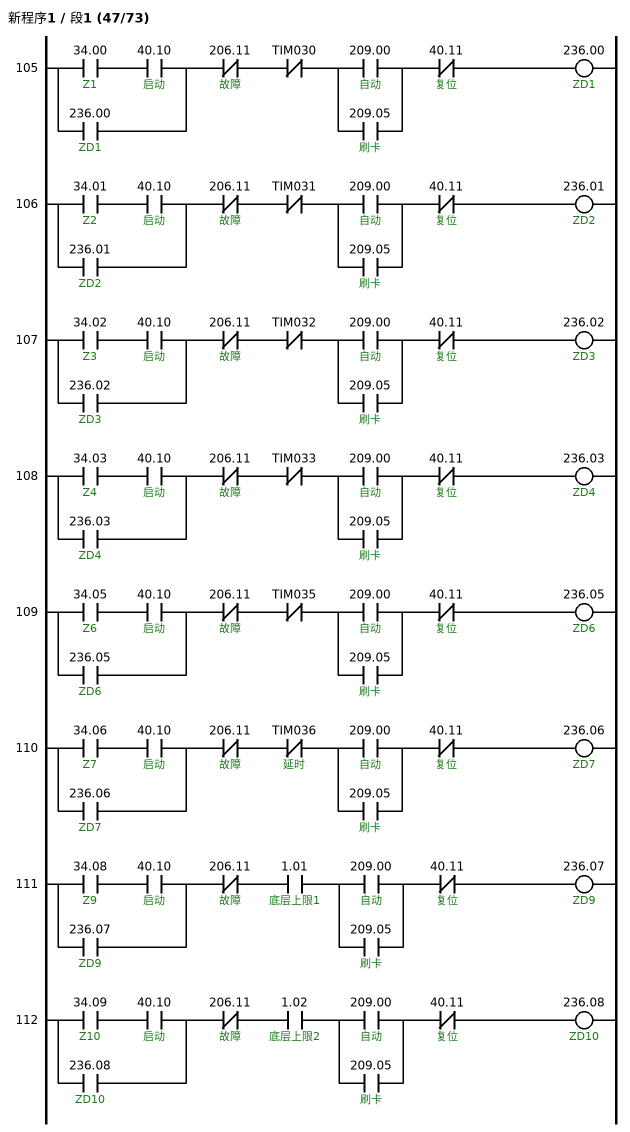
; [picture p48: 新程序1 / 段1, rungs 105-112]
; rung 105
LD 34.00  ; Z1
AND 40.10  ; 启动
OR 236.00  ; ZD1
ANDNOT 206.11  ; 故障
ANDNOT TIM030
LD 209.00  ; 自动
OR 209.05  ; 刷卡
ANDLD
ANDNOT 40.11  ; 复位
OUT 236.00  ; ZD1
; rung 106
LD 34.01  ; Z2
AND 40.10  ; 启动
OR 236.01  ; ZD2
ANDNOT 206.11  ; 故障
ANDNOT TIM031
LD 209.00  ; 自动
OR 209.05  ; 刷卡
ANDLD
ANDNOT 40.11  ; 复位
OUT 236.01  ; ZD2
; rung 107
LD 34.02  ; Z3
AND 40.10  ; 启动
OR 236.02  ; ZD3
ANDNOT 206.11  ; 故障
ANDNOT TIM032
LD 209.00  ; 自动
OR 209.05  ; 刷卡
ANDLD
ANDNOT 40.11  ; 复位
OUT 236.02  ; ZD3
; rung 108
LD 34.03  ; Z4
AND 40.10  ; 启动
OR 236.03  ; ZD4
ANDNOT 206.11  ; 故障
ANDNOT TIM033
LD 209.00  ; 自动
OR 209.05  ; 刷卡
ANDLD
ANDNOT 40.11  ; 复位
OUT 236.03  ; ZD4
; rung 109
LD 34.05  ; Z6
AND 40.10  ; 启动
OR 236.05  ; ZD6
ANDNOT 206.11  ; 故障
ANDNOT TIM035
LD 209.00  ; 自动
OR 209.05  ; 刷卡
ANDLD
ANDNOT 40.11  ; 复位
OUT 236.05  ; ZD6
; rung 110
LD 34.06  ; Z7
AND 40.10  ; 启动
OR 236.06  ; ZD7
ANDNOT 206.11  ; 故障
ANDNOT TIM036  ; 延时
LD 209.00  ; 自动
OR 209.05  ; 刷卡
ANDLD
ANDNOT 40.11  ; 复位
OUT 236.06  ; ZD7
; rung 111
LD 34.08  ; Z9
AND 40.10  ; 启动
OR 236.07  ; ZD9
ANDNOT 206.11  ; 故障
AND 1.01  ; 底层上限1
LD 209.00  ; 自动
OR 209.05  ; 刷卡
ANDLD
ANDNOT 40.11  ; 复位
OUT 236.07  ; ZD9
; rung 112
LD 34.09  ; Z10
AND 40.10  ; 启动
OR 236.08  ; ZD10
ANDNOT 206.11  ; 故障
AND 1.02  ; 底层上限2
LD 209.00  ; 自动
OR 209.05  ; 刷卡
ANDLD
ANDNOT 40.11  ; 复位
OUT 236.08  ; ZD10

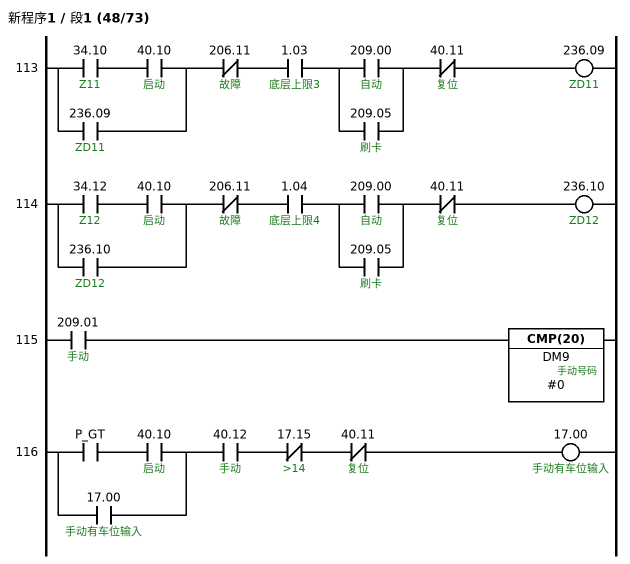
; rung 113
LD 34.10  ; Z11
AND 40.10  ; 启动
OR 236.09  ; ZD11
ANDNOT 206.11  ; 故障
AND 1.03  ; 底层上限3
LD 209.00  ; 自动
OR 209.05  ; 刷卡
ANDLD
ANDNOT 40.11  ; 复位
OUT 236.09  ; ZD11
; rung 114
LD 34.12  ; Z12
AND 40.10  ; 启动
OR 236.10  ; ZD12
ANDNOT 206.11  ; 故障
AND 1.04  ; 底层上限4
LD 209.00  ; 自动
OR 209.05  ; 刷卡
ANDLD
ANDNOT 40.11  ; 复位
OUT 236.10  ; ZD12
; rung 115
LD 209.01  ; 手动
CMP(20) DM9 #0  ; 手动号码
; rung 116
LD P_GT
AND 40.10  ; 启动
OR 17.00  ; 手动有车位输入
AND 40.12  ; 手动
ANDNOT 17.15  ; >14
ANDNOT 40.11  ; 复位
OUT 17.00  ; 手动有车位输入

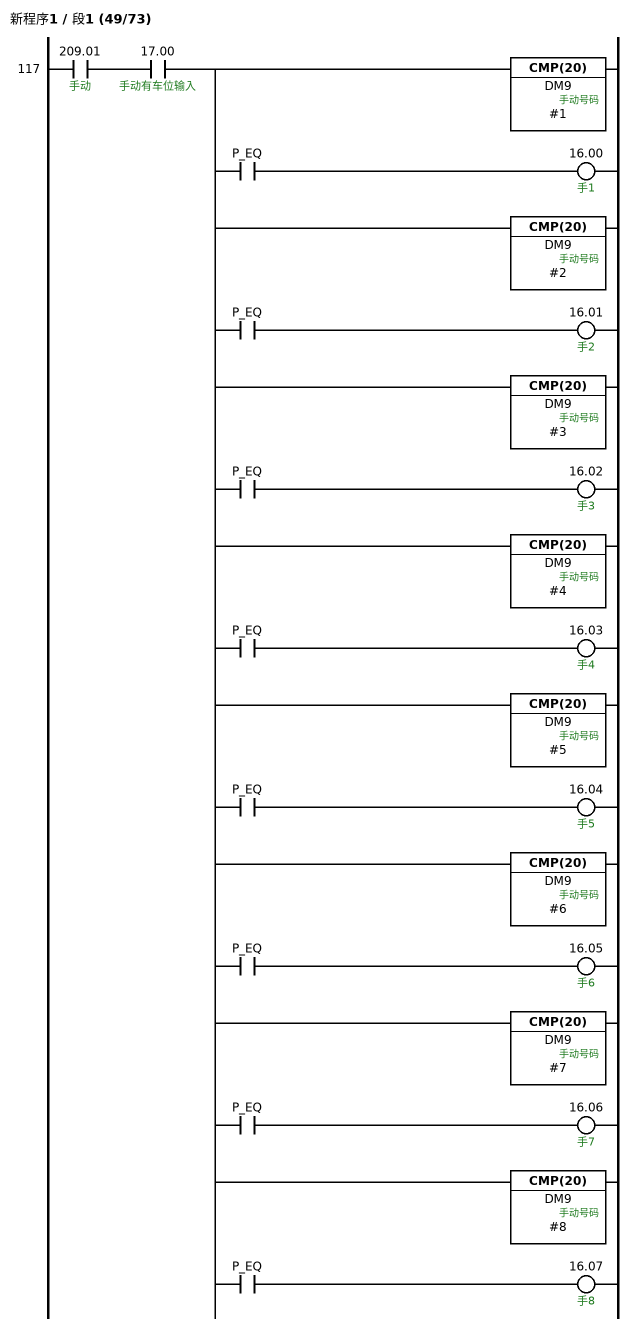

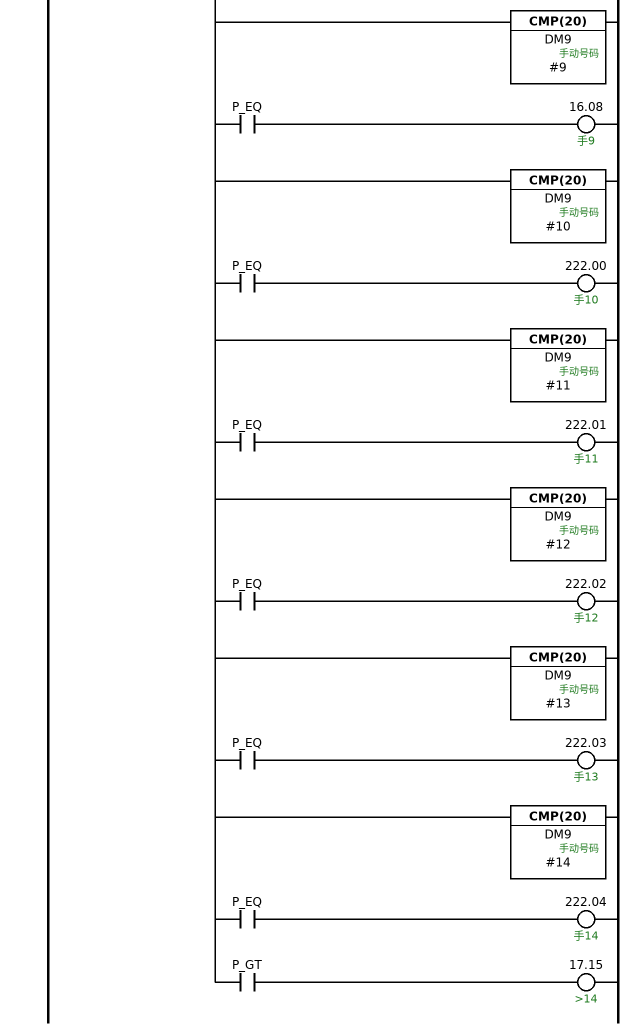
; rung 117
LD 209.01  ; 手动
AND 17.00  ; 手动有车位输入
OUT TR0
CMP(20) DM9 #1  ; 手动号码
AND P_EQ
OUT 16.00  ; 手1
LD TR0
CMP(20) DM9 #2  ; 手动号码
AND P_EQ
OUT 16.01  ; 手2
LD TR0
CMP(20) DM9 #3  ; 手动号码
AND P_EQ
OUT 16.02  ; 手3
LD TR0
CMP(20) DM9 #4  ; 手动号码
AND P_EQ
OUT 16.03  ; 手4
LD TR0
CMP(20) DM9 #5  ; 手动号码
AND P_EQ
OUT 16.04  ; 手5
LD TR0
CMP(20) DM9 #6  ; 手动号码
AND P_EQ
OUT 16.05  ; 手6
LD TR0
CMP(20) DM9 #7  ; 手动号码
AND P_EQ
OUT 16.06  ; 手7
LD TR0
CMP(20) DM9 #8  ; 手动号码
AND P_EQ
OUT 16.07  ; 手8
LD TR0
CMP(20) DM9 #9  ; 手动号码
AND P_EQ
OUT 16.08  ; 手9
LD TR0
CMP(20) DM9 #10  ; 手动号码
AND P_EQ
OUT 222.00  ; 手10
LD TR0
CMP(20) DM9 #11  ; 手动号码
AND P_EQ
OUT 222.01  ; 手11
LD TR0
CMP(20) DM9 #12  ; 手动号码
AND P_EQ
OUT 222.02  ; 手12
LD TR0
CMP(20) DM9 #13  ; 手动号码
AND P_EQ
OUT 222.03  ; 手13
LD TR0
CMP(20) DM9 #14  ; 手动号码
AND P_EQ
OUT 222.04  ; 手14
LD TR0
AND P_GT
OUT 17.15  ; >14

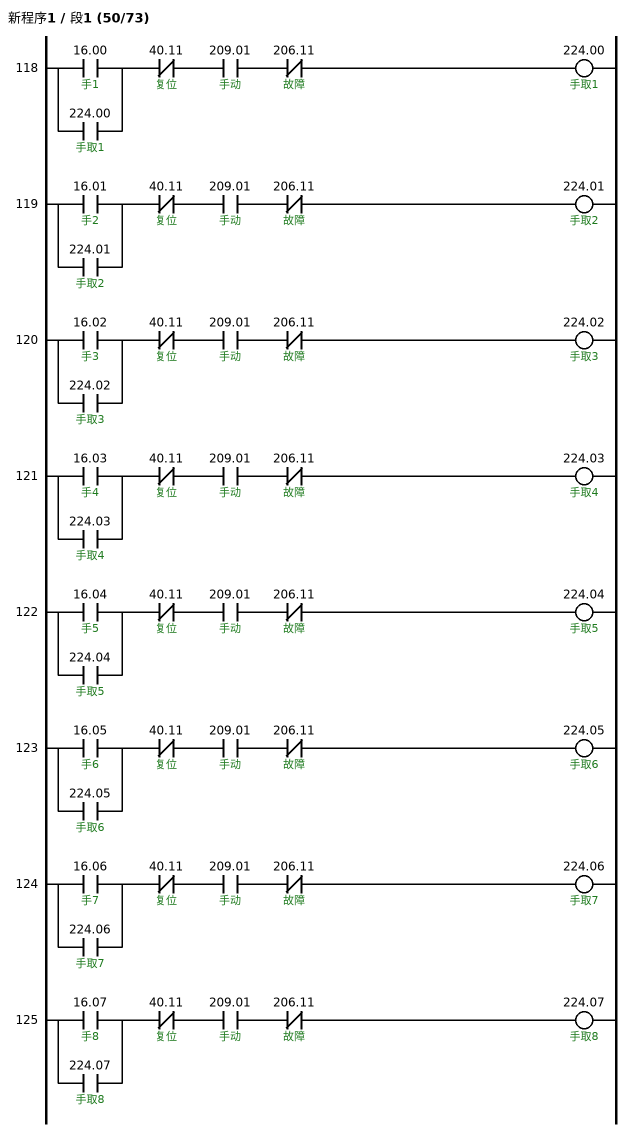
; rung 118
LD 16.00  ; 手1
OR 224.00  ; 手取1
ANDNOT 40.11  ; 复位
AND 209.01  ; 手动
ANDNOT 206.11  ; 故障
OUT 224.00  ; 手取1
; rung 119
LD 16.01  ; 手2
OR 224.01  ; 手取2
ANDNOT 40.11  ; 复位
AND 209.01  ; 手动
ANDNOT 206.11  ; 故障
OUT 224.01  ; 手取2
; rung 120
LD 16.02  ; 手3
OR 224.02  ; 手取3
ANDNOT 40.11  ; 复位
AND 209.01  ; 手动
ANDNOT 206.11  ; 故障
OUT 224.02  ; 手取3
; rung 121
LD 16.03  ; 手4
OR 224.03  ; 手取4
ANDNOT 40.11  ; 复位
AND 209.01  ; 手动
ANDNOT 206.11  ; 故障
OUT 224.03  ; 手取4
; rung 122
LD 16.04  ; 手5
OR 224.04  ; 手取5
ANDNOT 40.11  ; 复位
AND 209.01  ; 手动
ANDNOT 206.11  ; 故障
OUT 224.04  ; 手取5
; rung 123
LD 16.05  ; 手6
OR 224.05  ; 手取6
ANDNOT 40.11  ; 复位
AND 209.01  ; 手动
ANDNOT 206.11  ; 故障
OUT 224.05  ; 手取6
; rung 124
LD 16.06  ; 手7
OR 224.06  ; 手取7
ANDNOT 40.11  ; 复位
AND 209.01  ; 手动
ANDNOT 206.11  ; 故障
OUT 224.06  ; 手取7
; rung 125
LD 16.07  ; 手8
OR 224.07  ; 手取8
ANDNOT 40.11  ; 复位
AND 209.01  ; 手动
ANDNOT 206.11  ; 故障
OUT 224.07  ; 手取8

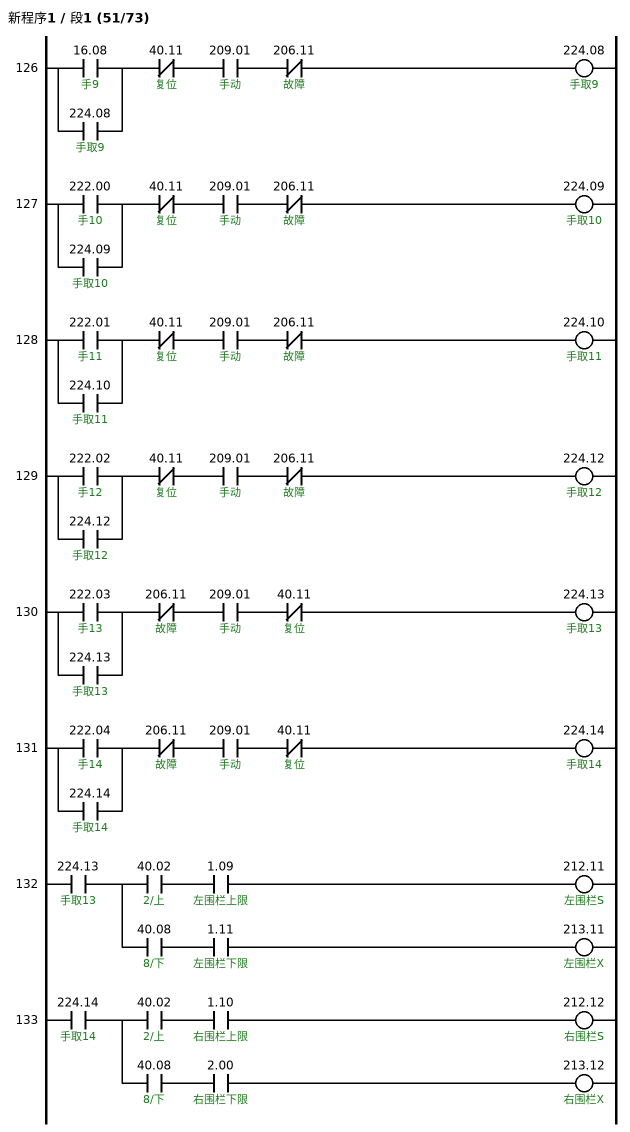
; rung 126
LD 16.08  ; 手9
OR 224.08  ; 手取9
ANDNOT 40.11  ; 复位
AND 209.01  ; 手动
ANDNOT 206.11  ; 故障
OUT 224.08  ; 手取9
; rung 127
LD 222.00  ; 手10
OR 224.09  ; 手取10
ANDNOT 40.11  ; 复位
AND 209.01  ; 手动
ANDNOT 206.11  ; 故障
OUT 224.09  ; 手取10
; rung 128
LD 222.01  ; 手11
OR 224.10  ; 手取11
ANDNOT 40.11  ; 复位
AND 209.01  ; 手动
ANDNOT 206.11  ; 故障
OUT 224.10  ; 手取11
; rung 129
LD 222.02  ; 手12
OR 224.12  ; 手取12
ANDNOT 40.11  ; 复位
AND 209.01  ; 手动
ANDNOT 206.11  ; 故障
OUT 224.12  ; 手取12
; rung 130
LD 222.03  ; 手13
OR 224.13  ; 手取13
ANDNOT 206.11  ; 故障
AND 209.01  ; 手动
ANDNOT 40.11  ; 复位
OUT 224.13  ; 手取13
; rung 131
LD 222.04  ; 手14
OR 224.14  ; 手取14
ANDNOT 206.11  ; 故障
AND 209.01  ; 手动
ANDNOT 40.11  ; 复位
OUT 224.14  ; 手取14
; rung 132
LD 224.13  ; 手取13
OUT TR0
AND 40.02  ; 2/上
AND 1.09  ; 左围栏上限
OUT 212.11  ; 左围栏S
LD TR0
AND 40.08  ; 8/下
AND 1.11  ; 左围栏下限
OUT 213.11  ; 左围栏X
; rung 133
LD 224.14  ; 手取14
OUT TR0
AND 40.02  ; 2/上
AND 1.10  ; 右围栏上限
OUT 212.12  ; 右围栏S
LD TR0
AND 40.08  ; 8/下
AND 2.00  ; 右围栏下限
OUT 213.12  ; 右围栏X

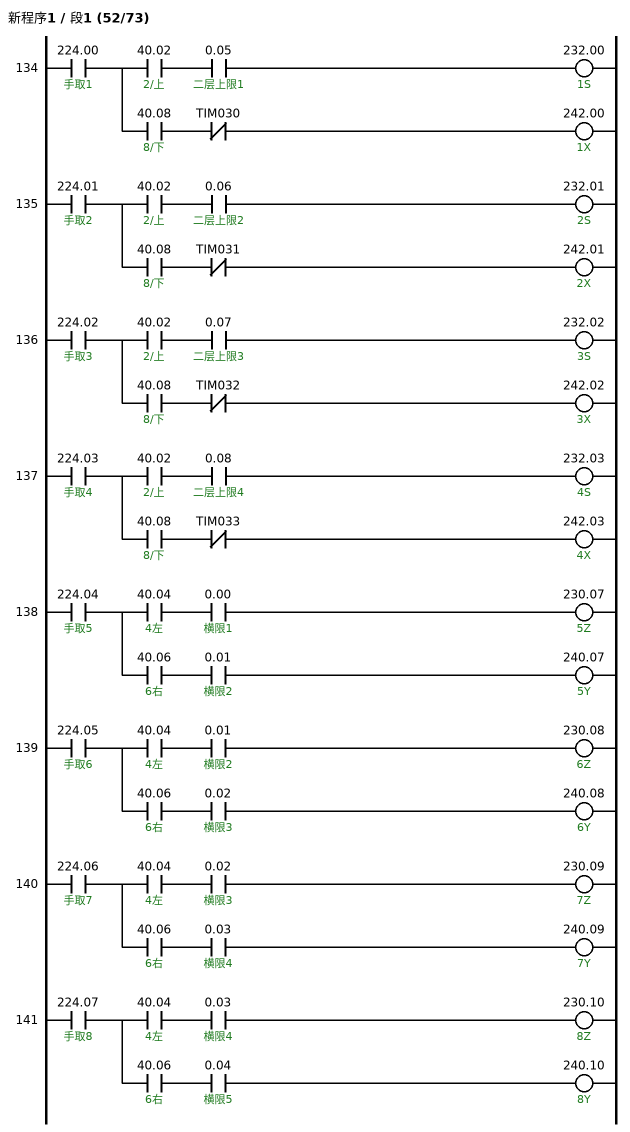
; rung 134
LD 224.00  ; 手取1
OUT TR0
AND 40.02  ; 2/上
AND 0.05  ; 二层上限1
OUT 232.00  ; 1S
LD TR0
AND 40.08  ; 8/下
ANDNOT TIM030
OUT 242.00  ; 1X
; rung 135
LD 224.01  ; 手取2
OUT TR0
AND 40.02  ; 2/上
AND 0.06  ; 二层上限2
OUT 232.01  ; 2S
LD TR0
AND 40.08  ; 8/下
ANDNOT TIM031
OUT 242.01  ; 2X
; rung 136
LD 224.02  ; 手取3
OUT TR0
AND 40.02  ; 2/上
AND 0.07  ; 二层上限3
OUT 232.02  ; 3S
LD TR0
AND 40.08  ; 8/下
ANDNOT TIM032
OUT 242.02  ; 3X
; rung 137
LD 224.03  ; 手取4
OUT TR0
AND 40.02  ; 2/上
AND 0.08  ; 二层上限4
OUT 232.03  ; 4S
LD TR0
AND 40.08  ; 8/下
ANDNOT TIM033
OUT 242.03  ; 4X
; rung 138
LD 224.04  ; 手取5
OUT TR0
AND 40.04  ; 4左
AND 0.00  ; 横限1
OUT 230.07  ; 5Z
LD TR0
AND 40.06  ; 6右
AND 0.01  ; 横限2
OUT 240.07  ; 5Y
; rung 139
LD 224.05  ; 手取6
OUT TR0
AND 40.04  ; 4左
AND 0.01  ; 横限2
OUT 230.08  ; 6Z
LD TR0
AND 40.06  ; 6右
AND 0.02  ; 横限3
OUT 240.08  ; 6Y
; rung 140
LD 224.06  ; 手取7
OUT TR0
AND 40.04  ; 4左
AND 0.02  ; 横限3
OUT 230.09  ; 7Z
LD TR0
AND 40.06  ; 6右
AND 0.03  ; 横限4
OUT 240.09  ; 7Y
; rung 141
LD 224.07  ; 手取8
OUT TR0
AND 40.04  ; 4左
AND 0.03  ; 横限4
OUT 230.10  ; 8Z
LD TR0
AND 40.06  ; 6右
AND 0.04  ; 横限5
OUT 240.10  ; 8Y

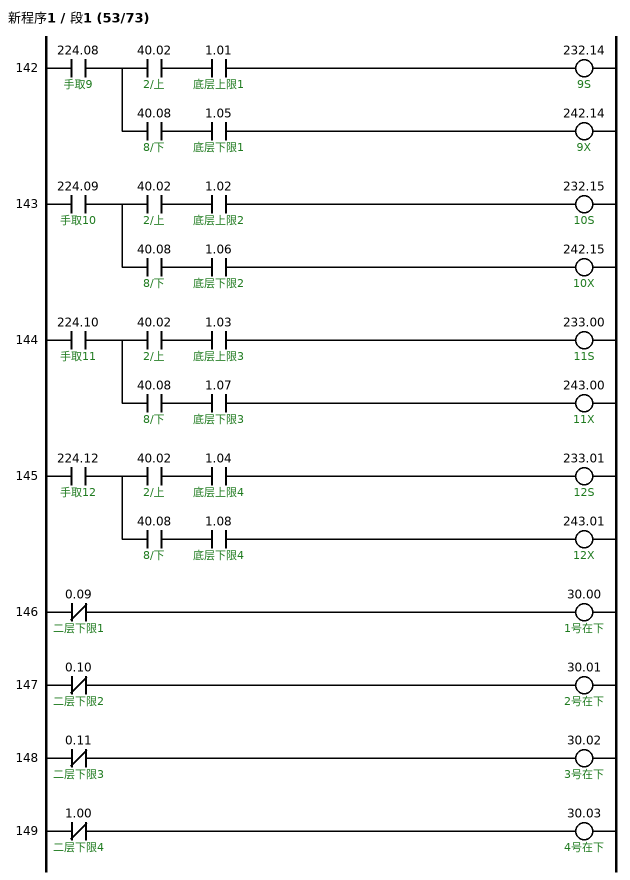
; rung 142
LD 224.08  ; 手取9
OUT TR0
AND 40.02  ; 2/上
AND 1.01  ; 底层上限1
OUT 232.14  ; 9S
LD TR0
AND 40.08  ; 8/下
AND 1.05  ; 底层下限1
OUT 242.14  ; 9X
; rung 143
LD 224.09  ; 手取10
OUT TR0
AND 40.02  ; 2/上
AND 1.02  ; 底层上限2
OUT 232.15  ; 10S
LD TR0
AND 40.08  ; 8/下
AND 1.06  ; 底层下限2
OUT 242.15  ; 10X
; rung 144
LD 224.10  ; 手取11
OUT TR0
AND 40.02  ; 2/上
AND 1.03  ; 底层上限3
OUT 233.00  ; 11S
LD TR0
AND 40.08  ; 8/下
AND 1.07  ; 底层下限3
OUT 243.00  ; 11X
; rung 145
LD 224.12  ; 手取12
OUT TR0
AND 40.02  ; 2/上
AND 1.04  ; 底层上限4
OUT 233.01  ; 12S
LD TR0
AND 40.08  ; 8/下
AND 1.08  ; 底层下限4
OUT 243.01  ; 12X
; rung 146
LDNOT 0.09  ; 二层下限1
OUT 30.00  ; 1号在下
; rung 147
LDNOT 0.10  ; 二层下限2
OUT 30.01  ; 2号在下
; rung 148
LDNOT 0.11  ; 二层下限3
OUT 30.02  ; 3号在下
; rung 149
LDNOT 1.00  ; 二层下限4
OUT 30.03  ; 4号在下

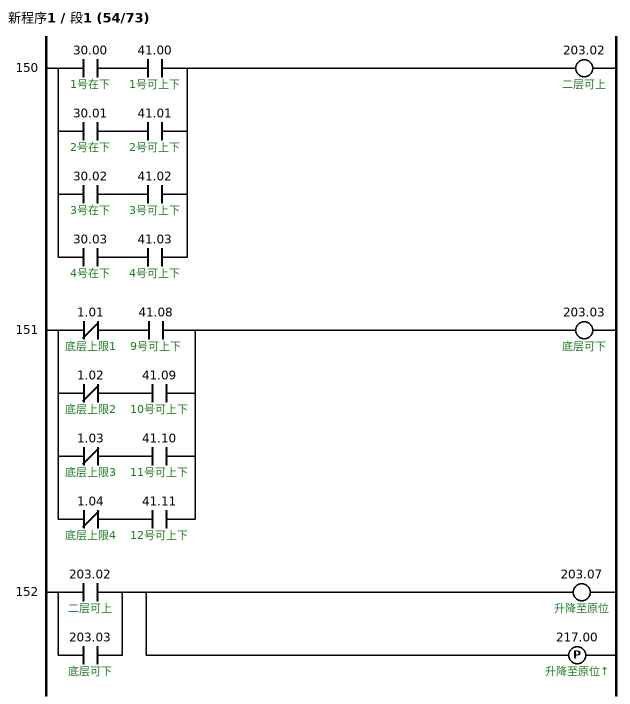
; rung 150
LD 30.00  ; 1号在下
AND 41.00  ; 1号可上下
LD 30.01  ; 2号在下
AND 41.01  ; 2号可上下
ORLD
LD 30.02  ; 3号在下
AND 41.02  ; 3号可上下
ORLD
LD 30.03  ; 4号在下
AND 41.03  ; 4号可上下
ORLD
OUT 203.02  ; 二层可上
; rung 151
LDNOT 1.01  ; 底层上限1
AND 41.08  ; 9号可上下
LDNOT 1.02  ; 底层上限2
AND 41.09  ; 10号可上下
ORLD
LDNOT 1.03  ; 底层上限3
AND 41.10  ; 11号可上下
ORLD
LDNOT 1.04  ; 底层上限4
AND 41.11  ; 12号可上下
ORLD
OUT 203.03  ; 底层可下
; rung 152
LD 203.02  ; 二层可上
OR 203.03  ; 底层可下
OUT 203.07  ; 升降至原位
DIFU(13) 217.00  ; 升降至原位↑

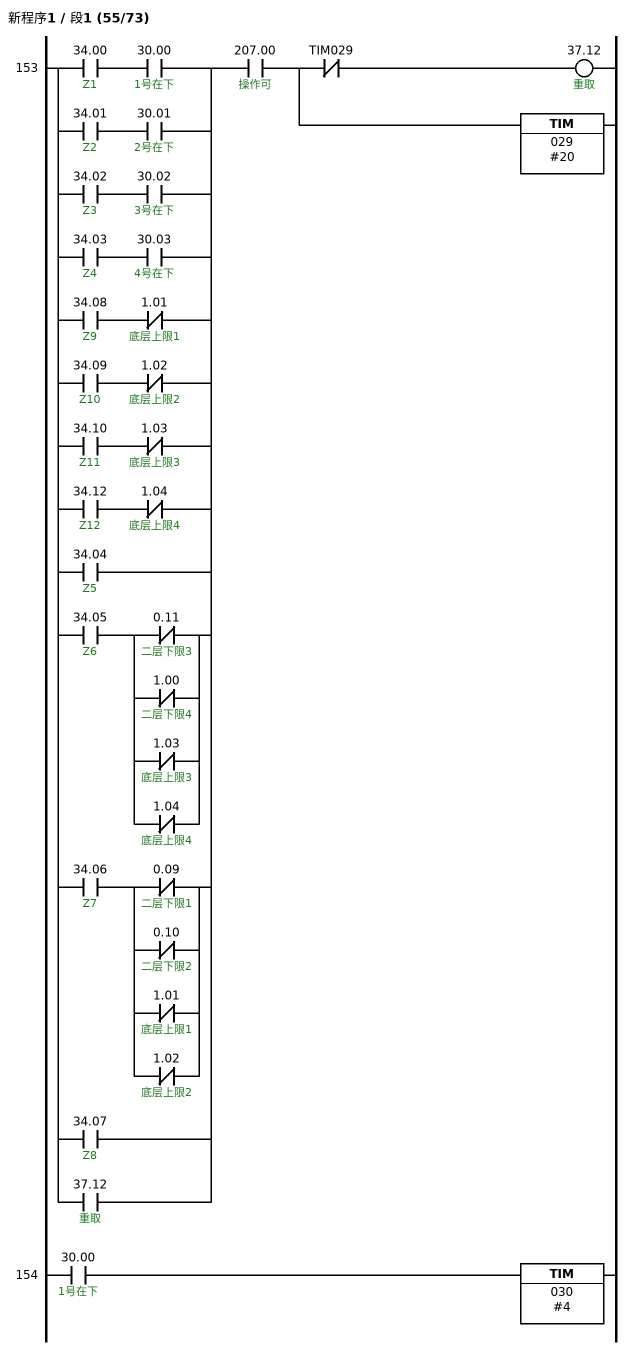
; rung 153
LD 34.00  ; Z1
AND 30.00  ; 1号在下
LD 34.01  ; Z2
AND 30.01  ; 2号在下
ORLD
LD 34.02  ; Z3
AND 30.02  ; 3号在下
ORLD
LD 34.03  ; Z4
AND 30.03  ; 4号在下
ORLD
LD 34.08  ; Z9
ANDNOT 1.01  ; 底层上限1
ORLD
LD 34.09  ; Z10
ANDNOT 1.02  ; 底层上限2
ORLD
LD 34.10  ; Z11
ANDNOT 1.03  ; 底层上限3
ORLD
LD 34.12  ; Z12
ANDNOT 1.04  ; 底层上限4
ORLD
OR 34.04  ; Z5
LD 34.05  ; Z6
LDNOT 0.11  ; 二层下限3
ORNOT 1.00  ; 二层下限4
ORNOT 1.03  ; 底层上限3
ORNOT 1.04  ; 底层上限4
ANDLD
ORLD
LD 34.06  ; Z7
LDNOT 0.09  ; 二层下限1
ORNOT 0.10  ; 二层下限2
ORNOT 1.01  ; 底层上限1
ORNOT 1.02  ; 底层上限2
ANDLD
ORLD
OR 34.07  ; Z8
OR 37.12  ; 重取
AND 207.00  ; 操作可
OUT TR0
ANDNOT TIM029
OUT 37.12  ; 重取
LD TR0
TIM 029 #20
; rung 154
LD 30.00  ; 1号在下
TIM 030 #4

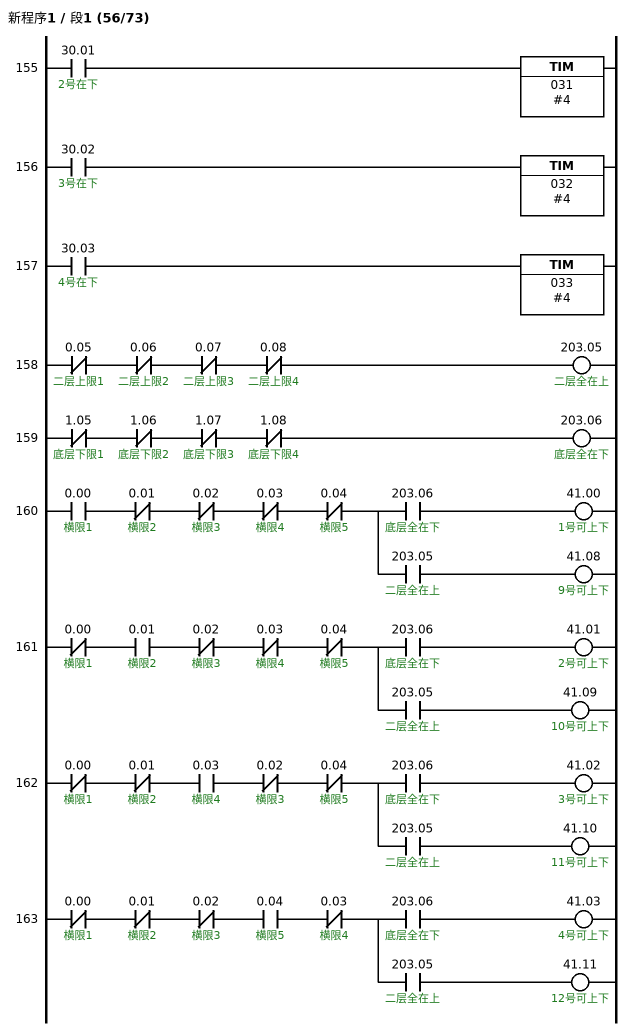
; rung 155
LD 30.01  ; 2号在下
TIM 031 #4
; rung 156
LD 30.02  ; 3号在下
TIM 032 #4
; rung 157
LD 30.03  ; 4号在下
TIM 033 #4
; rung 158
LDNOT 0.05  ; 二层上限1
ANDNOT 0.06  ; 二层上限2
ANDNOT 0.07  ; 二层上限3
ANDNOT 0.08  ; 二层上限4
OUT 203.05  ; 二层全在上
; rung 159
LDNOT 1.05  ; 底层下限1
ANDNOT 1.06  ; 底层下限2
ANDNOT 1.07  ; 底层下限3
ANDNOT 1.08  ; 底层下限4
OUT 203.06  ; 底层全在下
; rung 160
LD 0.00  ; 横限1
ANDNOT 0.01  ; 横限2
ANDNOT 0.02  ; 横限3
ANDNOT 0.03  ; 横限4
ANDNOT 0.04  ; 横限5
OUT TR0
AND 203.06  ; 底层全在下
OUT 41.00  ; 1号可上下
LD TR0
AND 203.05  ; 二层全在上
OUT 41.08  ; 9号可上下
; rung 161
LDNOT 0.00  ; 横限1
AND 0.01  ; 横限2
ANDNOT 0.02  ; 横限3
ANDNOT 0.03  ; 横限4
ANDNOT 0.04  ; 横限5
OUT TR0
AND 203.06  ; 底层全在下
OUT 41.01  ; 2号可上下
LD TR0
AND 203.05  ; 二层全在上
OUT 41.09  ; 10号可上下
; rung 162
LDNOT 0.00  ; 横限1
ANDNOT 0.01  ; 横限2
AND 0.03  ; 横限4
ANDNOT 0.02  ; 横限3
ANDNOT 0.04  ; 横限5
OUT TR0
AND 203.06  ; 底层全在下
OUT 41.02  ; 3号可上下
LD TR0
AND 203.05  ; 二层全在上
OUT 41.10  ; 11号可上下
; rung 163
LDNOT 0.00  ; 横限1
ANDNOT 0.01  ; 横限2
ANDNOT 0.02  ; 横限3
AND 0.04  ; 横限5
ANDNOT 0.03  ; 横限4
OUT TR0
AND 203.06  ; 底层全在下
OUT 41.03  ; 4号可上下
LD TR0
AND 203.05  ; 二层全在上
OUT 41.11  ; 12号可上下

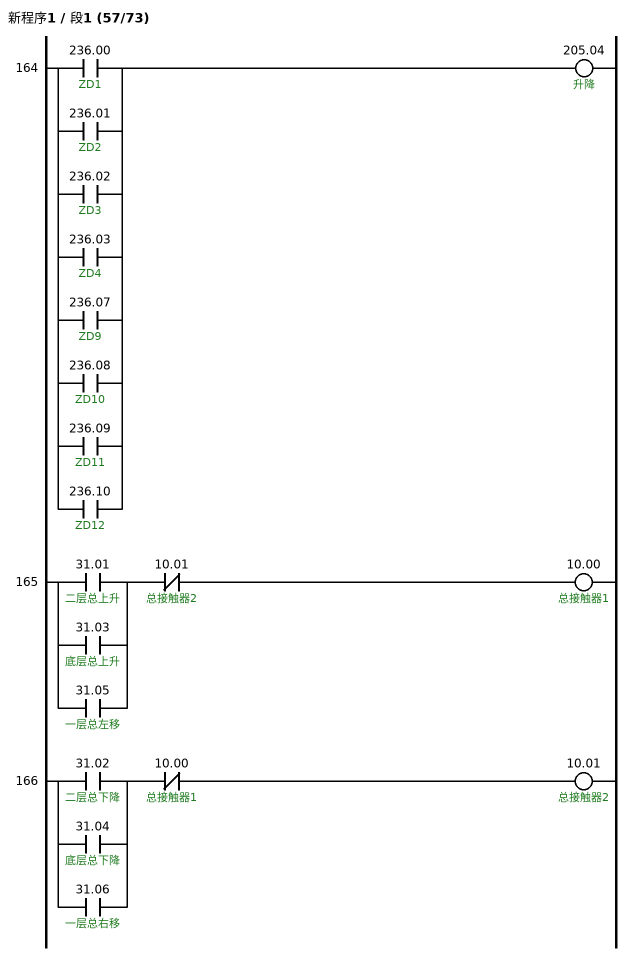
; rung 164
LD 236.00  ; ZD1
OR 236.01  ; ZD2
OR 236.02  ; ZD3
OR 236.03  ; ZD4
OR 236.07  ; ZD9
OR 236.08  ; ZD10
OR 236.09  ; ZD11
OR 236.10  ; ZD12
OUT 205.04  ; 升降
; rung 165
LD 31.01  ; 二层总上升
OR 31.03  ; 底层总上升
OR 31.05  ; 一层总左移
ANDNOT 10.01  ; 总接触器2
OUT 10.00  ; 总接触器1
; rung 166
LD 31.02  ; 二层总下降
OR 31.04  ; 底层总下降
OR 31.06  ; 一层总右移
ANDNOT 10.00  ; 总接触器1
OUT 10.01  ; 总接触器2

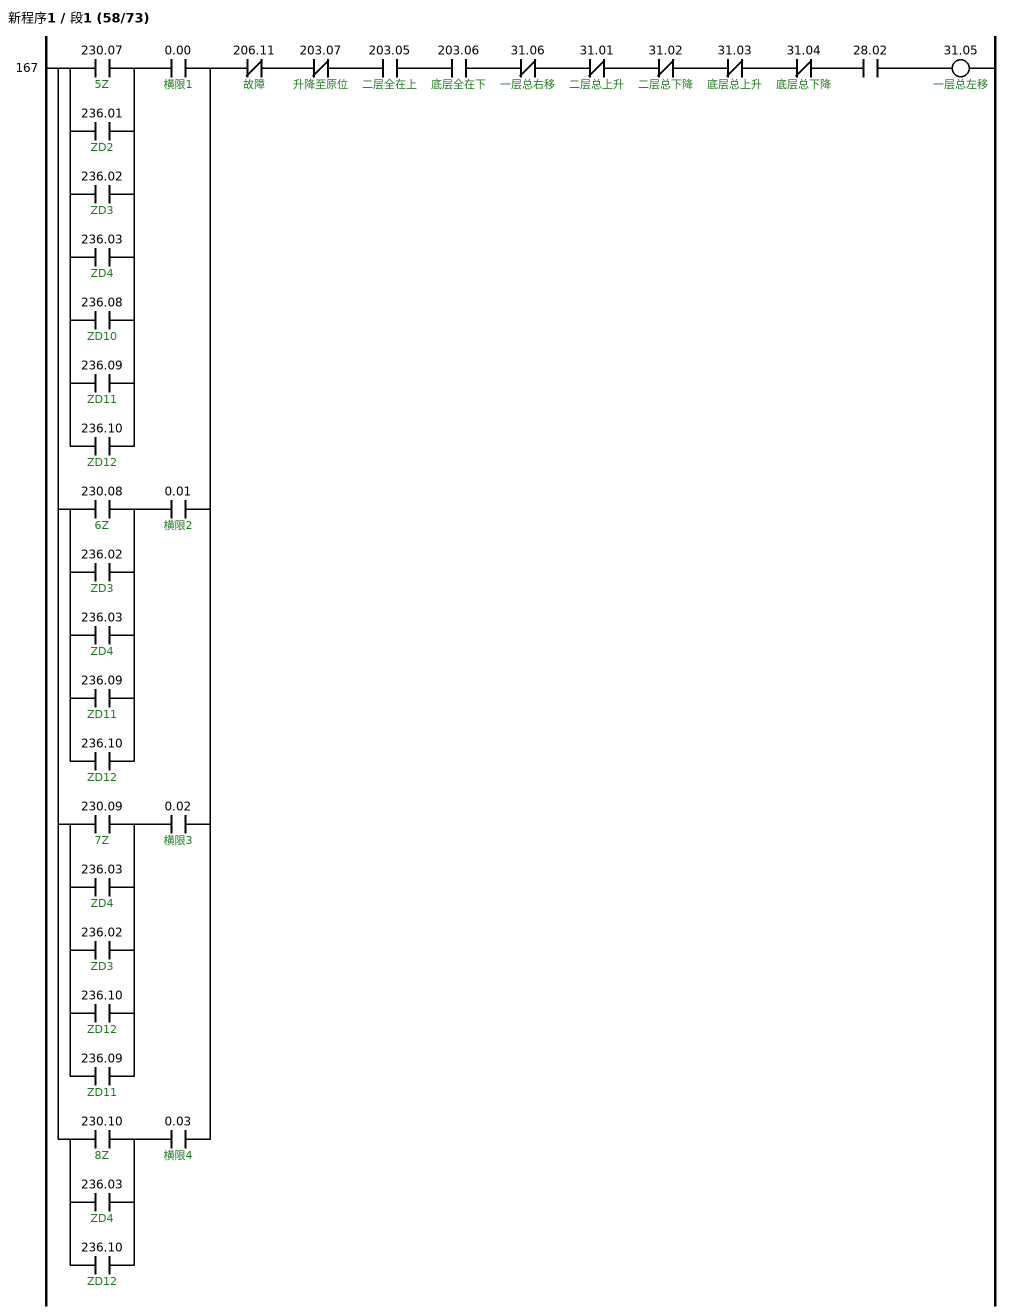
; rung 167
LD 230.07  ; 5Z
OR 236.01  ; ZD2
OR 236.02  ; ZD3
OR 236.03  ; ZD4
OR 236.08  ; ZD10
OR 236.09  ; ZD11
OR 236.10  ; ZD12
AND 0.00  ; 横限1
LD 230.08  ; 6Z
OR 236.02  ; ZD3
OR 236.03  ; ZD4
OR 236.09  ; ZD11
OR 236.10  ; ZD12
AND 0.01  ; 横限2
ORLD
LD 230.09  ; 7Z
OR 236.03  ; ZD4
OR 236.02  ; ZD3
OR 236.10  ; ZD12
OR 236.09  ; ZD11
AND 0.02  ; 横限3
ORLD
LD 230.10  ; 8Z
OR 236.03  ; ZD4
OR 236.10  ; ZD12
AND 0.03  ; 横限4
ORLD
ANDNOT 206.11  ; 故障
ANDNOT 203.07  ; 升降至原位
AND 203.05  ; 二层全在上
AND 203.06  ; 底层全在下
ANDNOT 31.06  ; 一层总右移
ANDNOT 31.01  ; 二层总上升
ANDNOT 31.02  ; 二层总下降
ANDNOT 31.03  ; 底层总上升
ANDNOT 31.04  ; 底层总下降
AND 28.02
OUT 31.05  ; 一层总左移

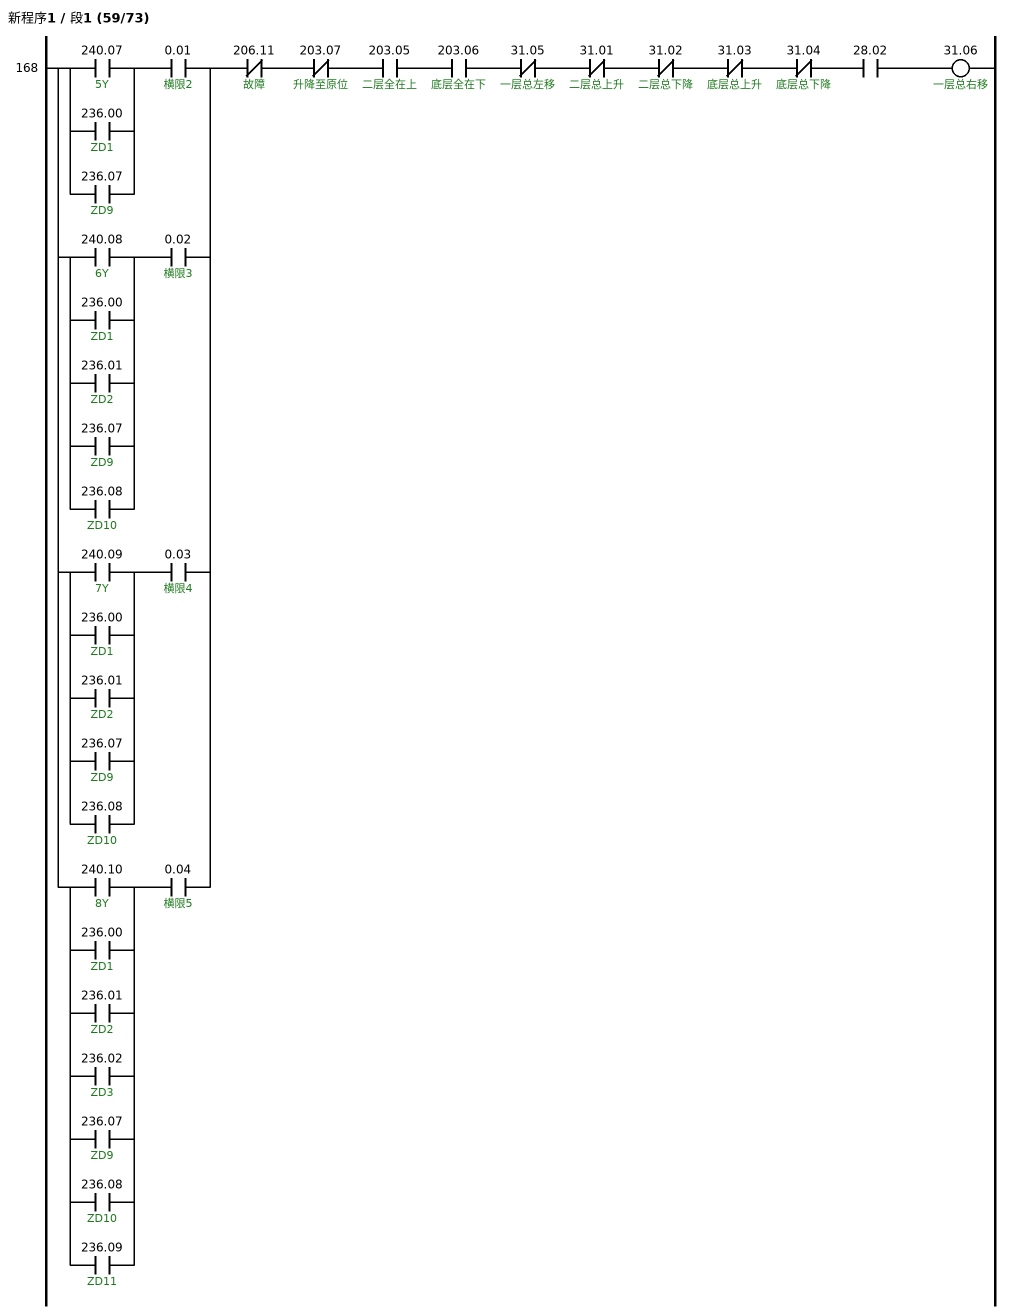
; rung 168
LD 240.07  ; 5Y
OR 236.00  ; ZD1
OR 236.07  ; ZD9
AND 0.01  ; 横限2
LD 240.08  ; 6Y
OR 236.00  ; ZD1
OR 236.01  ; ZD2
OR 236.07  ; ZD9
OR 236.08  ; ZD10
AND 0.02  ; 横限3
ORLD
LD 240.09  ; 7Y
OR 236.00  ; ZD1
OR 236.01  ; ZD2
OR 236.07  ; ZD9
OR 236.08  ; ZD10
AND 0.03  ; 横限4
ORLD
LD 240.10  ; 8Y
OR 236.00  ; ZD1
OR 236.01  ; ZD2
OR 236.02  ; ZD3
OR 236.07  ; ZD9
OR 236.08  ; ZD10
OR 236.09  ; ZD11
AND 0.04  ; 横限5
ORLD
ANDNOT 206.11  ; 故障
ANDNOT 203.07  ; 升降至原位
AND 203.05  ; 二层全在上
AND 203.06  ; 底层全在下
ANDNOT 31.05  ; 一层总左移
ANDNOT 31.01  ; 二层总上升
ANDNOT 31.02  ; 二层总下降
ANDNOT 31.03  ; 底层总上升
ANDNOT 31.04  ; 底层总下降
AND 28.02
OUT 31.06  ; 一层总右移

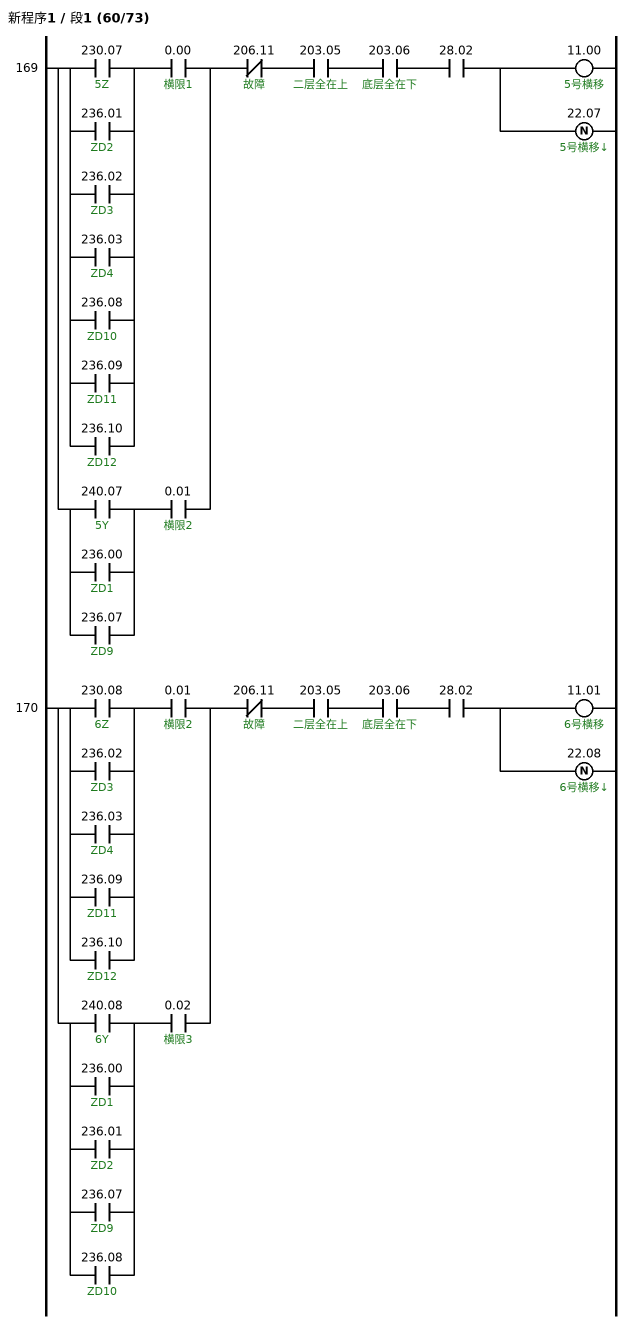
; rung 169
LD 230.07  ; 5Z
OR 236.01  ; ZD2
OR 236.02  ; ZD3
OR 236.03  ; ZD4
OR 236.08  ; ZD10
OR 236.09  ; ZD11
OR 236.10  ; ZD12
AND 0.00  ; 横限1
LD 240.07  ; 5Y
OR 236.00  ; ZD1
OR 236.07  ; ZD9
AND 0.01  ; 横限2
ORLD
ANDNOT 206.11  ; 故障
AND 203.05  ; 二层全在上
AND 203.06  ; 底层全在下
AND 28.02
OUT 11.00  ; 5号横移
DIFD(14) 22.07  ; 5号横移↓
; rung 170
LD 230.08  ; 6Z
OR 236.02  ; ZD3
OR 236.03  ; ZD4
OR 236.09  ; ZD11
OR 236.10  ; ZD12
AND 0.01  ; 横限2
LD 240.08  ; 6Y
OR 236.00  ; ZD1
OR 236.01  ; ZD2
OR 236.07  ; ZD9
OR 236.08  ; ZD10
AND 0.02  ; 横限3
ORLD
ANDNOT 206.11  ; 故障
AND 203.05  ; 二层全在上
AND 203.06  ; 底层全在下
AND 28.02
OUT 11.01  ; 6号横移
DIFD(14) 22.08  ; 6号横移↓

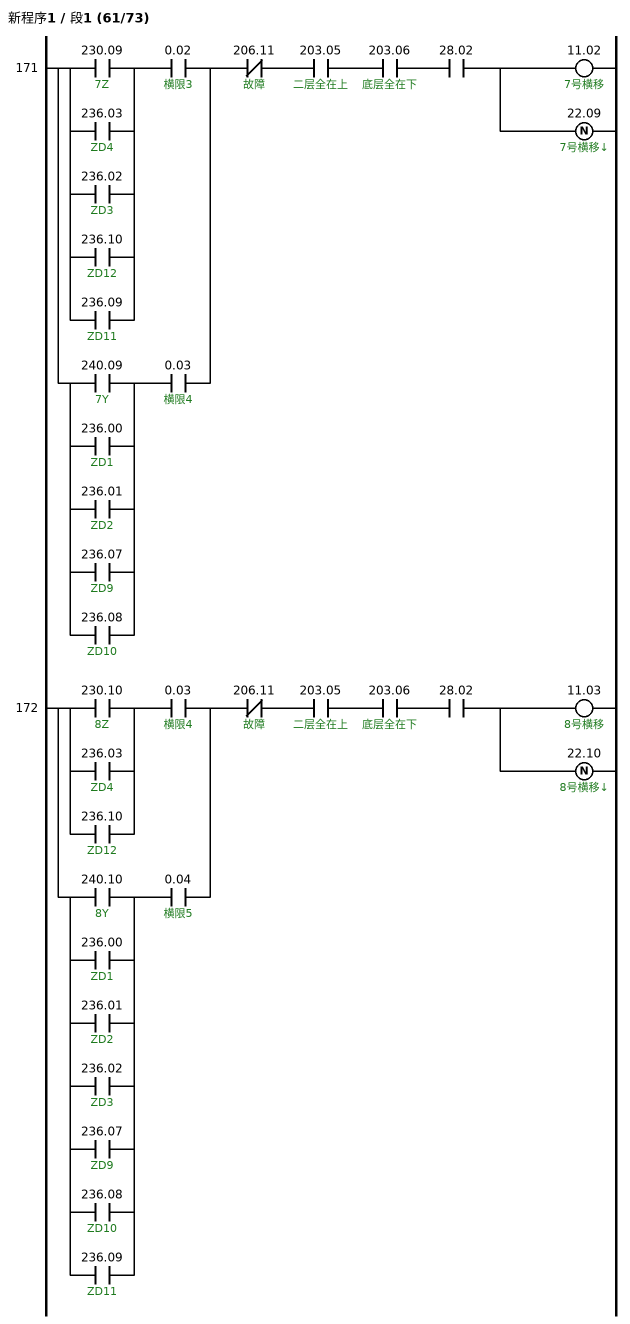
; rung 171
LD 230.09  ; 7Z
OR 236.03  ; ZD4
OR 236.02  ; ZD3
OR 236.10  ; ZD12
OR 236.09  ; ZD11
AND 0.02  ; 横限3
LD 240.09  ; 7Y
OR 236.00  ; ZD1
OR 236.01  ; ZD2
OR 236.07  ; ZD9
OR 236.08  ; ZD10
AND 0.03  ; 横限4
ORLD
ANDNOT 206.11  ; 故障
AND 203.05  ; 二层全在上
AND 203.06  ; 底层全在下
AND 28.02
OUT 11.02  ; 7号横移
DIFD(14) 22.09  ; 7号横移↓
; rung 172
LD 230.10  ; 8Z
OR 236.03  ; ZD4
OR 236.10  ; ZD12
AND 0.03  ; 横限4
LD 240.10  ; 8Y
OR 236.00  ; ZD1
OR 236.01  ; ZD2
OR 236.02  ; ZD3
OR 236.07  ; ZD9
OR 236.08  ; ZD10
OR 236.09  ; ZD11
AND 0.04  ; 横限5
ORLD
ANDNOT 206.11  ; 故障
AND 203.05  ; 二层全在上
AND 203.06  ; 底层全在下
AND 28.02
OUT 11.03  ; 8号横移
DIFD(14) 22.10  ; 8号横移↓

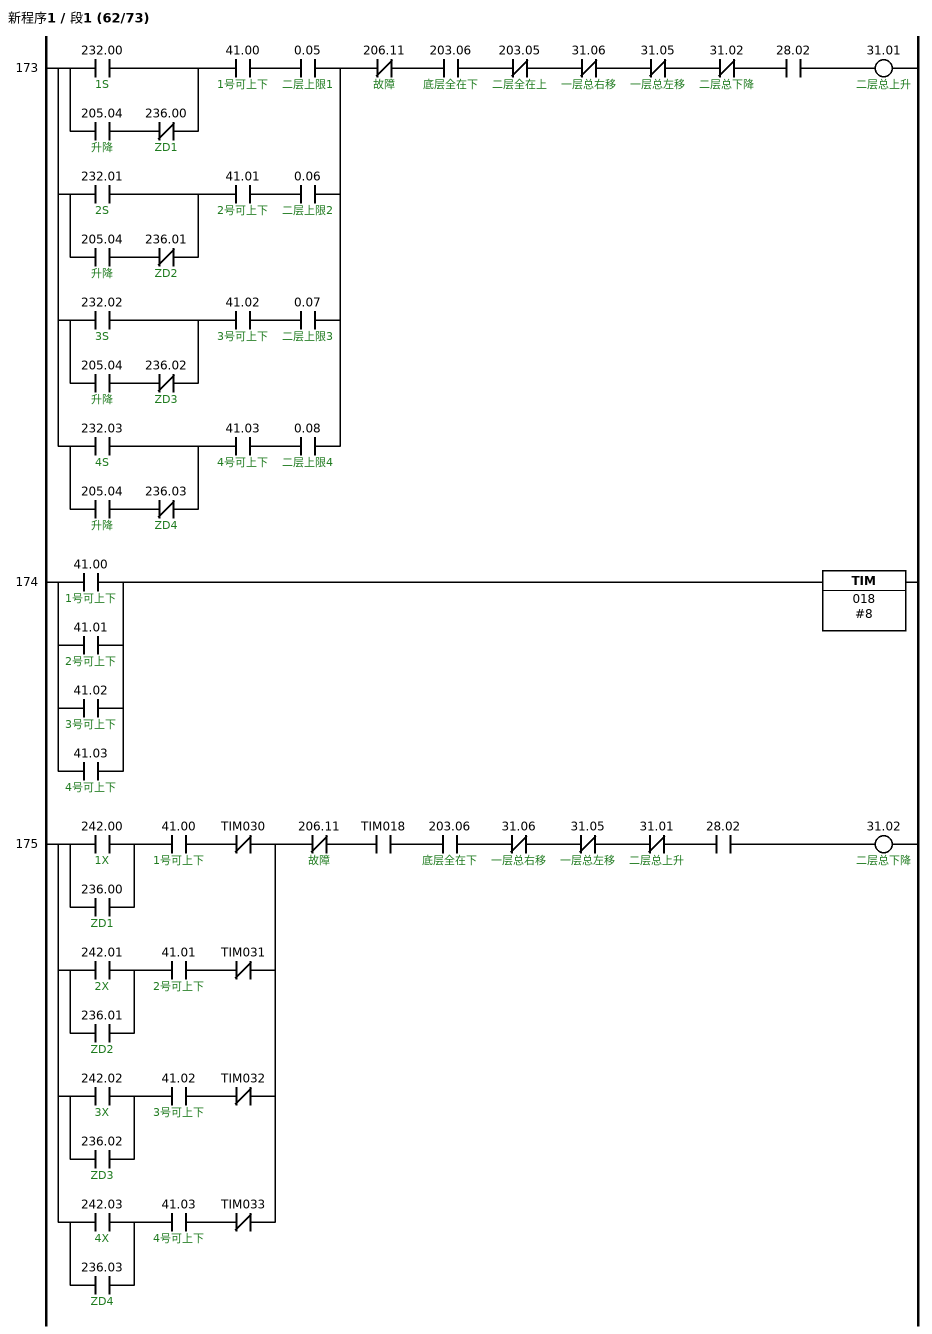
; rung 173
LD 232.00  ; 1S
LD 205.04  ; 升降
ANDNOT 236.00  ; ZD1
ORLD
AND 41.00  ; 1号可上下
AND 0.05  ; 二层上限1
LD 232.01  ; 2S
LD 205.04  ; 升降
ANDNOT 236.01  ; ZD2
ORLD
AND 41.01  ; 2号可上下
AND 0.06  ; 二层上限2
ORLD
LD 232.02  ; 3S
LD 205.04  ; 升降
ANDNOT 236.02  ; ZD3
ORLD
AND 41.02  ; 3号可上下
AND 0.07  ; 二层上限3
ORLD
LD 232.03  ; 4S
LD 205.04  ; 升降
ANDNOT 236.03  ; ZD4
ORLD
AND 41.03  ; 4号可上下
AND 0.08  ; 二层上限4
ORLD
ANDNOT 206.11  ; 故障
AND 203.06  ; 底层全在下
ANDNOT 203.05  ; 二层全在上
ANDNOT 31.06  ; 一层总右移
ANDNOT 31.05  ; 一层总左移
ANDNOT 31.02  ; 二层总下降
AND 28.02
OUT 31.01  ; 二层总上升
; rung 174
LD 41.00  ; 1号可上下
OR 41.01  ; 2号可上下
OR 41.02  ; 3号可上下
OR 41.03  ; 4号可上下
TIM 018 #8
; rung 175
LD 242.00  ; 1X
OR 236.00  ; ZD1
AND 41.00  ; 1号可上下
ANDNOT TIM030
LD 242.01  ; 2X
OR 236.01  ; ZD2
AND 41.01  ; 2号可上下
ANDNOT TIM031
ORLD
LD 242.02  ; 3X
OR 236.02  ; ZD3
AND 41.02  ; 3号可上下
ANDNOT TIM032
ORLD
LD 242.03  ; 4X
OR 236.03  ; ZD4
AND 41.03  ; 4号可上下
ANDNOT TIM033
ORLD
ANDNOT 206.11  ; 故障
AND TIM018
AND 203.06  ; 底层全在下
ANDNOT 31.06  ; 一层总右移
ANDNOT 31.05  ; 一层总左移
ANDNOT 31.01  ; 二层总上升
AND 28.02
OUT 31.02  ; 二层总下降

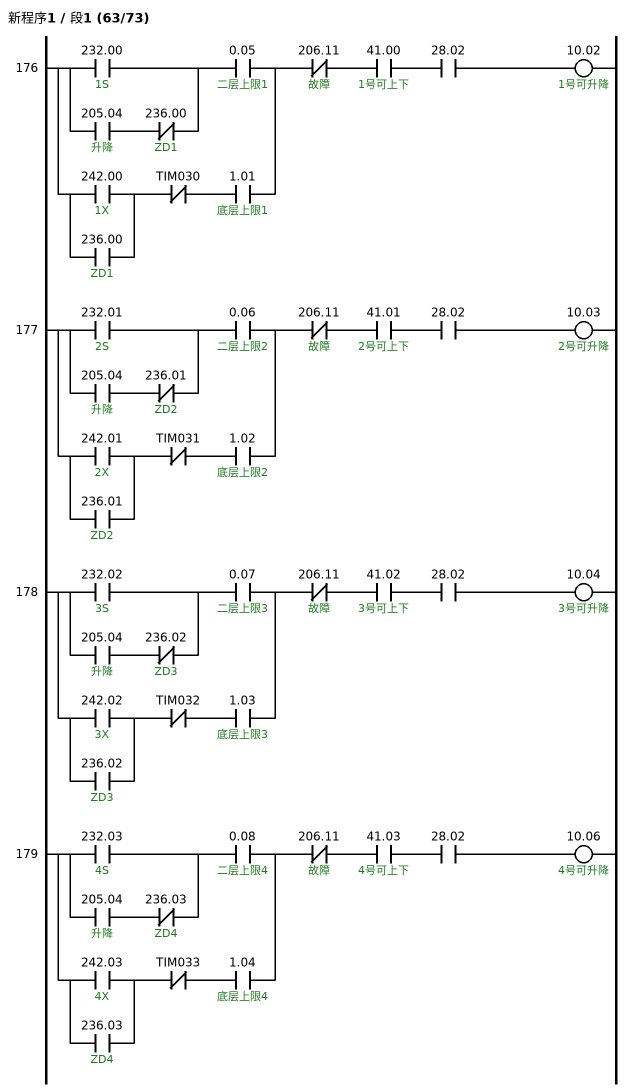
; rung 176
LD 232.00  ; 1S
LD 205.04  ; 升降
ANDNOT 236.00  ; ZD1
ORLD
AND 0.05  ; 二层上限1
LD 242.00  ; 1X
OR 236.00  ; ZD1
ANDNOT TIM030
AND 1.01  ; 底层上限1
ORLD
ANDNOT 206.11  ; 故障
AND 41.00  ; 1号可上下
AND 28.02
OUT 10.02  ; 1号可升降
; rung 177
LD 232.01  ; 2S
LD 205.04  ; 升降
ANDNOT 236.01  ; ZD2
ORLD
AND 0.06  ; 二层上限2
LD 242.01  ; 2X
OR 236.01  ; ZD2
ANDNOT TIM031
AND 1.02  ; 底层上限2
ORLD
ANDNOT 206.11  ; 故障
AND 41.01  ; 2号可上下
AND 28.02
OUT 10.03  ; 2号可升降
; rung 178
LD 232.02  ; 3S
LD 205.04  ; 升降
ANDNOT 236.02  ; ZD3
ORLD
AND 0.07  ; 二层上限3
LD 242.02  ; 3X
OR 236.02  ; ZD3
ANDNOT TIM032
AND 1.03  ; 底层上限3
ORLD
ANDNOT 206.11  ; 故障
AND 41.02  ; 3号可上下
AND 28.02
OUT 10.04  ; 3号可升降
; rung 179
LD 232.03  ; 4S
LD 205.04  ; 升降
ANDNOT 236.03  ; ZD4
ORLD
AND 0.08  ; 二层上限4
LD 242.03  ; 4X
OR 236.03  ; ZD4
ANDNOT TIM033
AND 1.04  ; 底层上限4
ORLD
ANDNOT 206.11  ; 故障
AND 41.03  ; 4号可上下
AND 28.02
OUT 10.06  ; 4号可升降

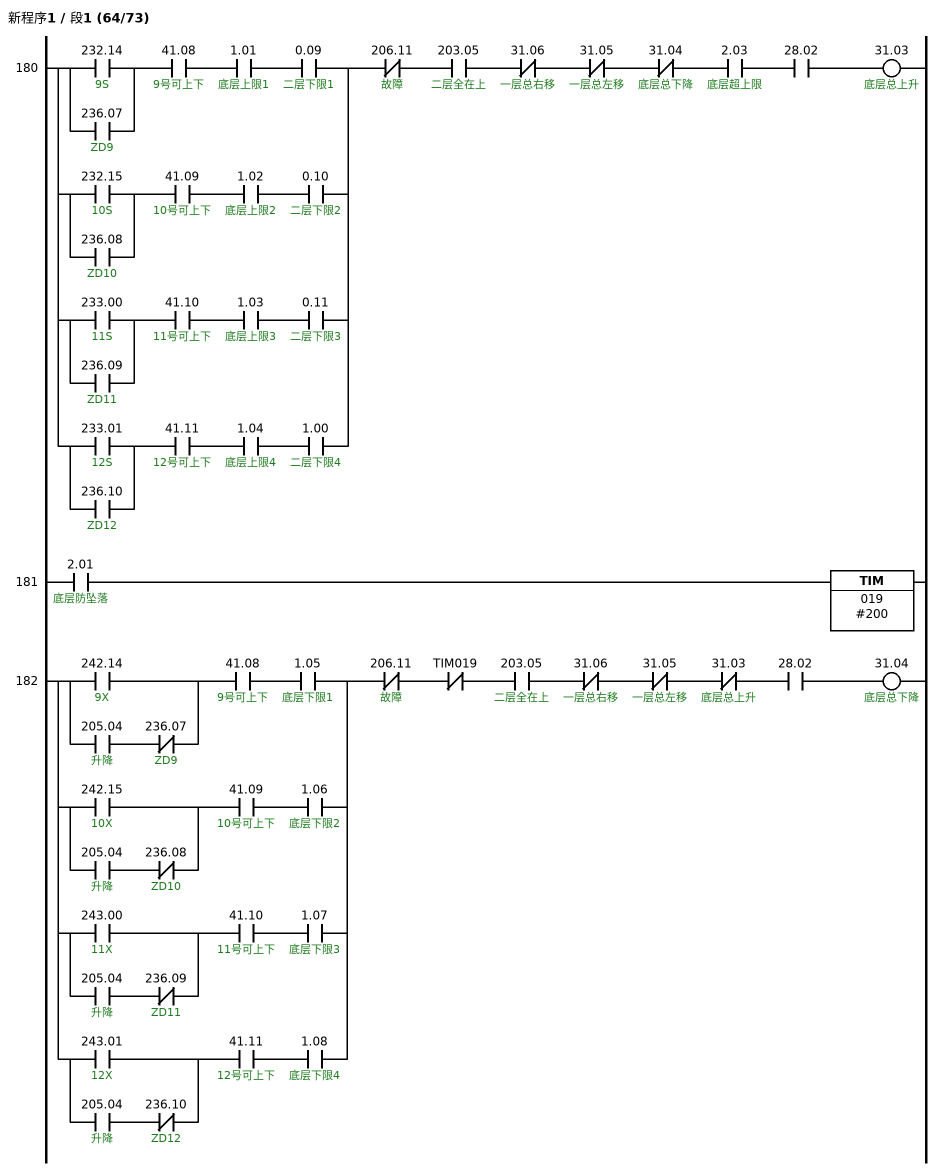
; rung 180
LD 232.14  ; 9S
OR 236.07  ; ZD9
AND 41.08  ; 9号可上下
AND 1.01  ; 底层上限1
AND 0.09  ; 二层下限1
LD 232.15  ; 10S
OR 236.08  ; ZD10
AND 41.09  ; 10号可上下
AND 1.02  ; 底层上限2
AND 0.10  ; 二层下限2
ORLD
LD 233.00  ; 11S
OR 236.09  ; ZD11
AND 41.10  ; 11号可上下
AND 1.03  ; 底层上限3
AND 0.11  ; 二层下限3
ORLD
LD 233.01  ; 12S
OR 236.10  ; ZD12
AND 41.11  ; 12号可上下
AND 1.04  ; 底层上限4
AND 1.00  ; 二层下限4
ORLD
ANDNOT 206.11  ; 故障
AND 203.05  ; 二层全在上
ANDNOT 31.06  ; 一层总右移
ANDNOT 31.05  ; 一层总左移
ANDNOT 31.04  ; 底层总下降
AND 2.03  ; 底层超上限
AND 28.02
OUT 31.03  ; 底层总上升
; rung 181
LD 2.01  ; 底层防坠落
TIM 019 #200
; rung 182
LD 242.14  ; 9X
LD 205.04  ; 升降
ANDNOT 236.07  ; ZD9
ORLD
AND 41.08  ; 9号可上下
AND 1.05  ; 底层下限1
LD 242.15  ; 10X
LD 205.04  ; 升降
ANDNOT 236.08  ; ZD10
ORLD
AND 41.09  ; 10号可上下
AND 1.06  ; 底层下限2
ORLD
LD 243.00  ; 11X
LD 205.04  ; 升降
ANDNOT 236.09  ; ZD11
ORLD
AND 41.10  ; 11号可上下
AND 1.07  ; 底层下限3
ORLD
LD 243.01  ; 12X
LD 205.04  ; 升降
ANDNOT 236.10  ; ZD12
ORLD
AND 41.11  ; 12号可上下
AND 1.08  ; 底层下限4
ORLD
ANDNOT 206.11  ; 故障
ANDNOT TIM019
AND 203.05  ; 二层全在上
ANDNOT 31.06  ; 一层总右移
ANDNOT 31.05  ; 一层总左移
ANDNOT 31.03  ; 底层总上升
AND 28.02
OUT 31.04  ; 底层总下降

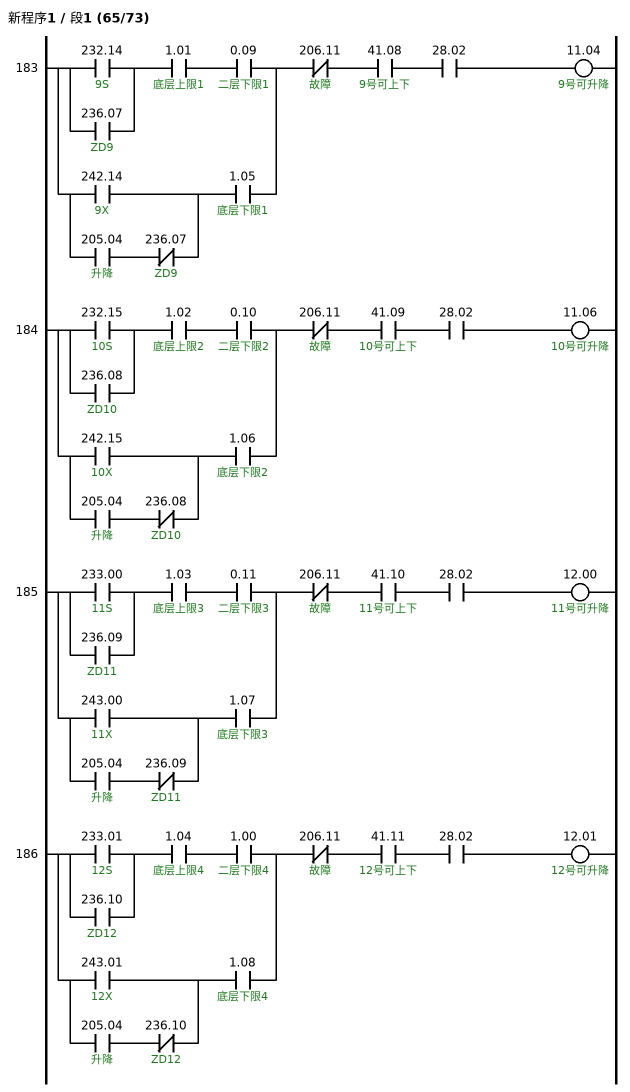
; rung 183
LD 232.14  ; 9S
OR 236.07  ; ZD9
AND 1.01  ; 底层上限1
AND 0.09  ; 二层下限1
LD 242.14  ; 9X
LD 205.04  ; 升降
ANDNOT 236.07  ; ZD9
ORLD
AND 1.05  ; 底层下限1
ORLD
ANDNOT 206.11  ; 故障
AND 41.08  ; 9号可上下
AND 28.02
OUT 11.04  ; 9号可升降
; rung 184
LD 232.15  ; 10S
OR 236.08  ; ZD10
AND 1.02  ; 底层上限2
AND 0.10  ; 二层下限2
LD 242.15  ; 10X
LD 205.04  ; 升降
ANDNOT 236.08  ; ZD10
ORLD
AND 1.06  ; 底层下限2
ORLD
ANDNOT 206.11  ; 故障
AND 41.09  ; 10号可上下
AND 28.02
OUT 11.06  ; 10号可升降
; rung 185
LD 233.00  ; 11S
OR 236.09  ; ZD11
AND 1.03  ; 底层上限3
AND 0.11  ; 二层下限3
LD 243.00  ; 11X
LD 205.04  ; 升降
ANDNOT 236.09  ; ZD11
ORLD
AND 1.07  ; 底层下限3
ORLD
ANDNOT 206.11  ; 故障
AND 41.10  ; 11号可上下
AND 28.02
OUT 12.00  ; 11号可升降
; rung 186
LD 233.01  ; 12S
OR 236.10  ; ZD12
AND 1.04  ; 底层上限4
AND 1.00  ; 二层下限4
LD 243.01  ; 12X
LD 205.04  ; 升降
ANDNOT 236.10  ; ZD12
ORLD
AND 1.08  ; 底层下限4
ORLD
ANDNOT 206.11  ; 故障
AND 41.11  ; 12号可上下
AND 28.02
OUT 12.01  ; 12号可升降

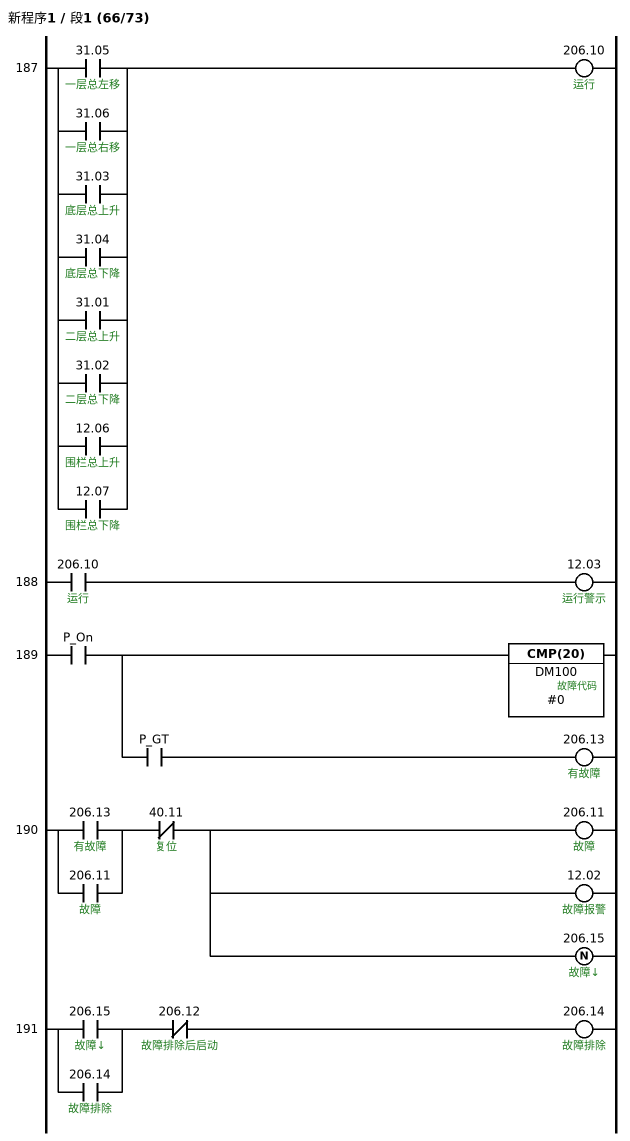
; rung 187
LD 31.05  ; 一层总左移
OR 31.06  ; 一层总右移
OR 31.03  ; 底层总上升
OR 31.04  ; 底层总下降
OR 31.01  ; 二层总上升
OR 31.02  ; 二层总下降
OR 12.06  ; 围栏总上升
OR 12.07  ; 围栏总下降
OUT 206.10  ; 运行
; rung 188
LD 206.10  ; 运行
OUT 12.03  ; 运行警示
; rung 189
LD P_On
CMP(20) DM100 #0  ; 故障代码
AND P_GT
OUT 206.13  ; 有故障
; rung 190
LD 206.13  ; 有故障
OR 206.11  ; 故障
ANDNOT 40.11  ; 复位
OUT 206.11  ; 故障
OUT 12.02  ; 故障报警
DIFD(14) 206.15  ; 故障↓
; rung 191
LD 206.15  ; 故障↓
OR 206.14  ; 故障排除
ANDNOT 206.12  ; 故障排除后启动
OUT 206.14  ; 故障排除

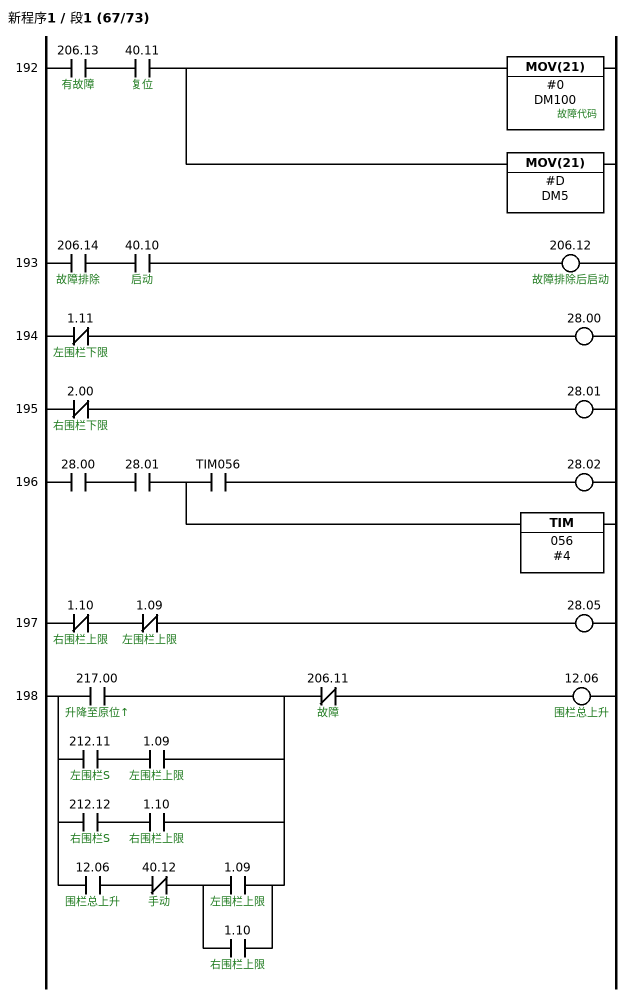
; rung 192
LD 206.13  ; 有故障
AND 40.11  ; 复位
MOV(21) #0 DM100  ; 故障代码
MOV(21) #D DM5
; rung 193
LD 206.14  ; 故障排除
AND 40.10  ; 启动
OUT 206.12  ; 故障排除后启动
; rung 194
LDNOT 1.11  ; 左围栏下限
OUT 28.00
; rung 195
LDNOT 2.00  ; 右围栏下限
OUT 28.01
; rung 196
LD 28.00
AND 28.01
OUT TR0
AND TIM056
OUT 28.02
LD TR0
TIM 056 #4
; rung 197
LDNOT 1.10  ; 右围栏上限
ANDNOT 1.09  ; 左围栏上限
OUT 28.05
; rung 198
LD 217.00  ; 升降至原位↑
LD 212.11  ; 左围栏S
AND 1.09  ; 左围栏上限
ORLD
LD 212.12  ; 右围栏S
AND 1.10  ; 右围栏上限
ORLD
LD 12.06  ; 围栏总上升
ANDNOT 40.12  ; 手动
LD 1.09  ; 左围栏上限
OR 1.10  ; 右围栏上限
ANDLD
ORLD
ANDNOT 206.11  ; 故障
OUT 12.06  ; 围栏总上升

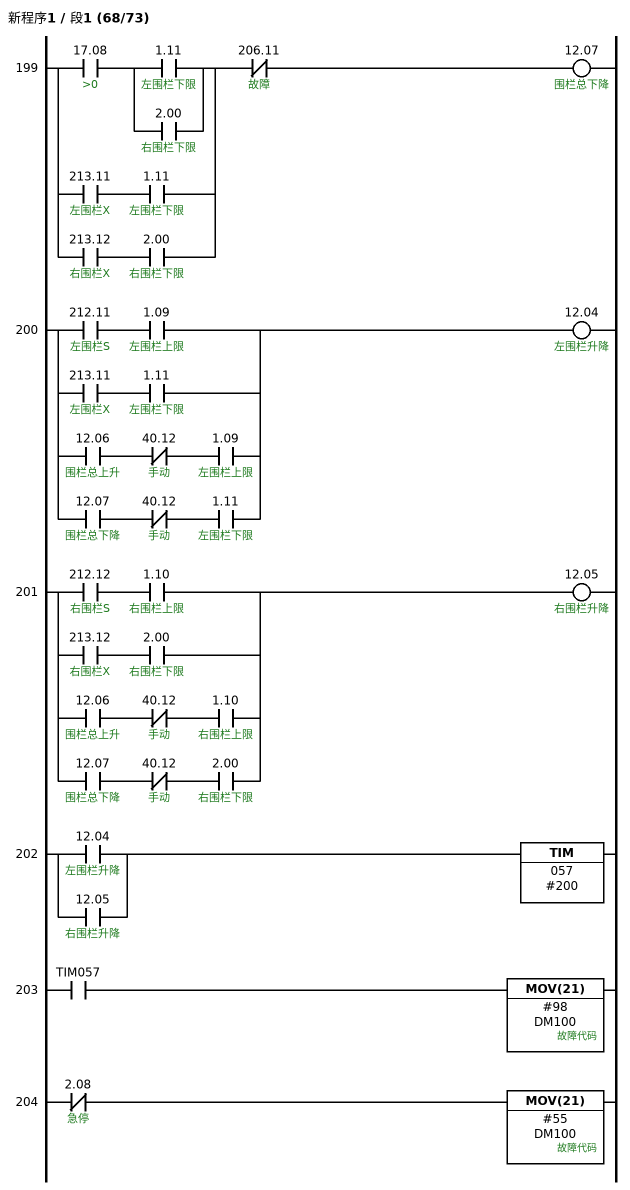
; rung 199
LD 17.08  ; >0
LD 1.11  ; 左围栏下限
OR 2.00  ; 右围栏下限
ANDLD
LD 213.11  ; 左围栏X
AND 1.11  ; 左围栏下限
ORLD
LD 213.12  ; 右围栏X
AND 2.00  ; 右围栏下限
ORLD
ANDNOT 206.11  ; 故障
OUT 12.07  ; 围栏总下降
; rung 200
LD 212.11  ; 左围栏S
AND 1.09  ; 左围栏上限
LD 213.11  ; 左围栏X
AND 1.11  ; 左围栏下限
ORLD
LD 12.06  ; 围栏总上升
ANDNOT 40.12  ; 手动
AND 1.09  ; 左围栏上限
ORLD
LD 12.07  ; 围栏总下降
ANDNOT 40.12  ; 手动
AND 1.11  ; 左围栏下限
ORLD
OUT 12.04  ; 左围栏升降
; rung 201
LD 212.12  ; 右围栏S
AND 1.10  ; 右围栏上限
LD 213.12  ; 右围栏X
AND 2.00  ; 右围栏下限
ORLD
LD 12.06  ; 围栏总上升
ANDNOT 40.12  ; 手动
AND 1.10  ; 右围栏上限
ORLD
LD 12.07  ; 围栏总下降
ANDNOT 40.12  ; 手动
AND 2.00  ; 右围栏下限
ORLD
OUT 12.05  ; 右围栏升降
; rung 202
LD 12.04  ; 左围栏升降
OR 12.05  ; 右围栏升降
TIM 057 #200
; rung 203
LD TIM057
MOV(21) #98 DM100  ; 故障代码
; rung 204
LDNOT 2.08  ; 急停
MOV(21) #55 DM100  ; 故障代码

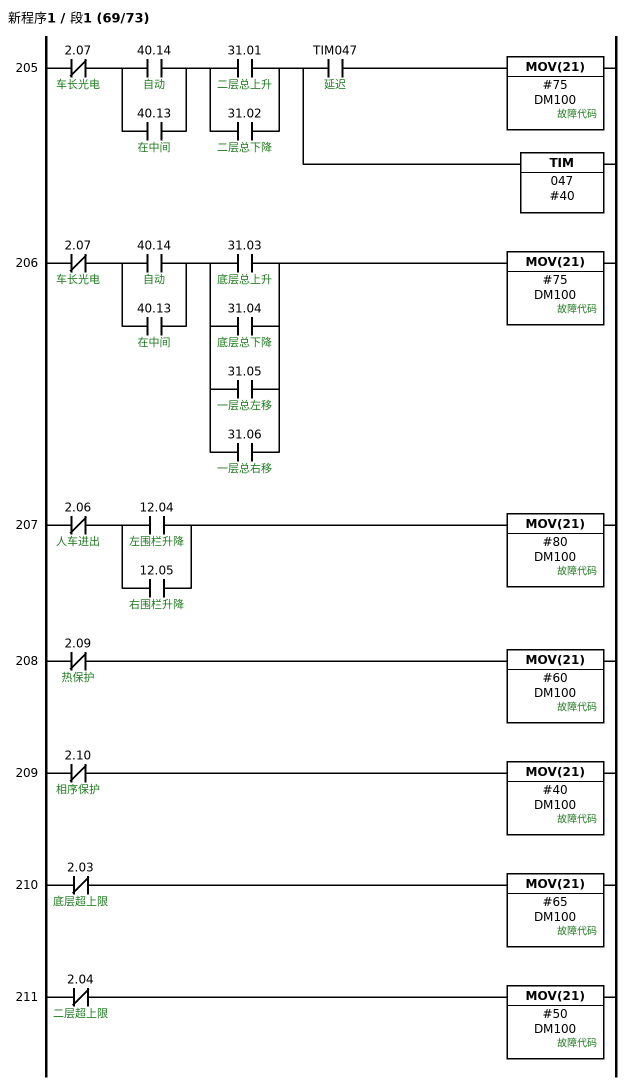
; rung 205
LDNOT 2.07  ; 车长光电
LD 40.14  ; 自动
OR 40.13  ; 在中间
ANDLD
LD 31.01  ; 二层总上升
OR 31.02  ; 二层总下降
ANDLD
OUT TR0
AND TIM047  ; 延迟
MOV(21) #75 DM100  ; 故障代码
LD TR0
TIM 047 #40
; rung 206
LDNOT 2.07  ; 车长光电
LD 40.14  ; 自动
OR 40.13  ; 在中间
ANDLD
LD 31.03  ; 底层总上升
OR 31.04  ; 底层总下降
OR 31.05  ; 一层总左移
OR 31.06  ; 一层总右移
ANDLD
MOV(21) #75 DM100  ; 故障代码
; rung 207
LDNOT 2.06  ; 人车进出
LD 12.04  ; 左围栏升降
OR 12.05  ; 右围栏升降
ANDLD
MOV(21) #80 DM100  ; 故障代码
; rung 208
LDNOT 2.09  ; 热保护
MOV(21) #60 DM100  ; 故障代码
; rung 209
LDNOT 2.10  ; 相序保护
MOV(21) #40 DM100  ; 故障代码
; rung 210
LDNOT 2.03  ; 底层超上限
MOV(21) #65 DM100  ; 故障代码
; rung 211
LDNOT 2.04  ; 二层超上限
MOV(21) #50 DM100  ; 故障代码

